TYPE CAN_TxMsgSlot :
STRUCT
	cobId : UINT;
    data  : ARRAY[0..7] OF USINT;
END_STRUCT
END_TYPE

(* stored: Version 1.1.0.1
   DUT CAN_TxMsgSlot: Id {e2d4410a-4abe-4a2a-8e75-cbf1e294c437} *)
